INTERFACE I_ErrorSubject

END_INTERFACE

(* stored: Version 1.1.0.1, ProductVersion 3.1.4024.13
   Itf I_ErrorSubject: Id {511cba63-e6c4-491a-88e6-04a1fcfdda57} *)
